FUNCTION_BLOCK SUBL_3_OK (* 3-variable data subscriber *)
  (* Standard: 61499-2 *)
  (* Version 1.0, 21-03-12, GASR, Universidade do Estado de Santa Catarina *)
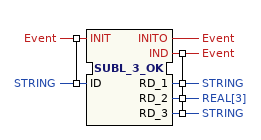
  EVENT_INPUT
    INIT WITH ID; (* Service initiaization *)
  END_EVENT
  EVENT_OUTPUT
    INITO; (* Initialization confirm *)
    IND WITH RD_1, RD_2, RD_3; (* Service indication *)
  END_EVENT
  VAR_INPUT
    ID : STRING; (* Default id is the FB instance name *)
  END_VAR
  VAR_OUTPUT
    RD_1 : STRING;
    RD_2 : ARRAY [0..2] OF REAL; (* Machine Position *)
    RD_3 : STRING; (* Current tool *)
  END_VAR
  SERVICE PUBL_3_OK/SUBL_3_OK (* Data publication service *)
    SEQUENCE normal_establishment
      PUBL_3_OK.INIT(ID) -> PUBL_3_OK.INITO();
      SUBL_3_OK.INIT(ID) -> SUBL_3_OK.INITO();
    END_SEQUENCE
    SEQUENCE normal_data_transfer
      PUBL_3_OK.REQ(SD_1,SD_2,SD_3) -> SUBL_3_OK.IND(RD_1,RD_2,RD_3);
    END_SEQUENCE
  END_SERVICE
END_FUNCTION_BLOCK
